FUNCTION_BLOCK PUBLISH_6 (* 6-Variable Publisher *)
  (* Standard: 61499-1; Classification: Communications *)
  (* Version 0.0, 2004-06-09, JHC, Rockwell Automation *)
  (* Compiler header: package fb.rt.net; *)
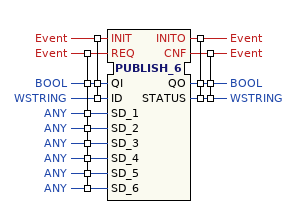
  EVENT_INPUT
    INIT WITH QI, ID; (* Service Initialization *)
    REQ WITH QI, SD_1, SD_2, SD_3, SD_4, SD_5, SD_6; (* Service Request *)
  END_EVENT
  EVENT_OUTPUT
    INITO WITH QO, STATUS; (* Initialization Confirm *)
    CNF WITH QO, STATUS; (* Service Confirmation *)
  END_EVENT
  VAR_INPUT
    QI : BOOL; (* Event Input Qualifier *)
    ID : WSTRING; (* Connection Identifier *)
    SD_1 : ANY; (* Data to Send *)
    SD_2 : ANY;
    SD_3 : ANY;
    SD_4 : ANY;
    SD_5 : ANY;
    SD_6 : ANY;
  END_VAR
  VAR_OUTPUT
    QO : BOOL; (* Event Output Qualifier *)
    STATUS : WSTRING; (* Service Status *)
  END_VAR
END_FUNCTION_BLOCK
